TYPE ST_IotProps :
STRUCT
	sName		: STRING;
	sValue		: STRING(2000);
	eUpdate 	: eUpdate;
	st_RW		: ST_RW;
	pAdress		: PVOID;
	diSize		: DINT;
	ClassType : __SYSTEM.TYPE_CLASS;
	bNumber		: BOOL;
	bJson		: BOOL;
END_STRUCT
END_TYPE

(* stored: Version 1.1.0.1, ProductVersion 3.1.4026.18
   DUT ST_IotProps: Id {b31f5181-60e6-48e8-9436-1680af4e776d} *)
